{attribute 'linkalways'} 
{attribute 'no_explicit_call' := 'This FB is a CLASS and must be accessed using methods or properties'}
{attribute 'enable_dynamic_creation'}
FUNCTION_BLOCK FINAL OR_BYTE EXTENDS Node
VAR
	in1 : _BYTE(0);
	in2 : _BYTE(0);
	out : _BYTE(0);
END_VAR

METHOD PUBLIC Clone : I_Node
VAR
	pNode : POINTER TO OR_BYTE;
END_VAR
pNode := __NEW(OR_BYTE);
Clone := pNode^;
END_METHOD

METHOD FB_init : BOOL
VAR_INPUT
	bInitRetains : BOOL; // if TRUE, the retain variables are initialized (warm start / cold start)
	bInCopyCode : BOOL;  // if TRUE, the instance afterwards gets moved into the copy code (online change)
END_VAR
AddInput('in1',THIS^.in1);
AddInput('in2',THIS^.in2);
AddOutput('out', THIS^.out);
END_METHOD

METHOD PROTECTED OnExecute
VAR
END_VAR
out.Value := in1.Value OR in2.Value;
END_METHOD

END_FUNCTION_BLOCK

(* stored: Version 1.1.0.1, ProductVersion 3.1.4024.15
   POU OR_BYTE: Id {b5fd27a2-c61d-4a75-a5d7-dc99798ad637}, SpecialFunc None
   Folder Constructor: Id {f5ef50de-7c03-4508-9dcc-0302c82d4ec9}
   Method Clone: Id {47b07a23-9b41-4ac3-922e-ce3342b2a216}
   Method FB_init: Id {2bc7ea9e-ad5c-409b-b4f9-79d8468fc2d2}
   Method OnExecute: Id {8e0a03bd-c195-4ba0-b565-795266d2ed03} *)
